DATA_BLOCK "FB_HGU_Motor_Control_Simple_DB"
{ S7_Optimized_Access := 'TRUE' }
VERSION : 1.0
NON_RETAIN
"FB_HGU_Motor_Control_Simple"

BEGIN

END_DATA_BLOCK